// TIA Portal V16 export
// export: Created 2024-12-03T15:41:45.7340631Z, ExportSetting WithReadOnly, DisplayName Totally Integrated Automation Portal, DisplayVersion V16 Update 6, DisplayName TIA Portal Version Control Interface, DisplayVersion V16 Update 2, DisplayName TIA Portal Openness, DisplayVersion V16 Update 6, DisplayName TIA Portal Teamcenter Gateway, DisplayVersion V16, DisplayName SINAMICS Startdrive Advanced, DisplayVersion V16 Update 5, DisplayName SINAMICS Startdrive G130, G150, S120, S150, SINAMICS MV, S210, DisplayVersion V16 Update 5, DisplayName SINAMICS Startdrive G110M, G120, G120C, G120D, G120P, G115D, DisplayVersion V16 Update 5, DisplayName STEP 7 Professional, DisplayVersion V16 Update 6, DisplayName STEP 7 Safety, DisplayVersion V16, DisplayName WinCC Advanced / Unified PC, DisplayVersion V16 Update 6
TYPE "Nord_Drive_UDT"
// stored: CreationDate 2023-04-19T11:30:38.0051651Z, InterfaceModifiedDate 2023-04-19T12:03:36.1263348Z, IsConsistent true, LibraryConformanceStatus The object is library-conformant., ModifiedDate 2023-04-19T12:03:36.1263348Z
   STRUCT
      Cmd : Struct   // MotorCommands
         Reset : Bool;
         OnAuto : Bool;
         OnManual : Bool;
         DirectionAuto : Bool;
         DirectionManual : Bool;
         SpeedAuto : Real;
         SpeedManual : Real;
         Interlock : Bool;
      END_STRUCT;
      Alarms : Struct
         NotOnTImedOut : "HmiAlarm";   // Motor not on in time
         NotOffTimedOut : "HmiAlarm";   // Motor not off in time
         ErrorFromDrive : "HmiAlarm";   // Error from drive
         CannotStartError : "HmiAlarm";   // Cannot start error
         EmergencyStopActive : "HmiAlarm";   // Emergency stop is active
         Disconnected : "HmiAlarm";   // The device is not connected
         WarningFromDrive { S7_SetPoint := 'True'} : "HmiAlarm";   // Warning from drive
         AlarmStatus : Word;   // lsb 0 not on | lsb 1 not off | lsb 2 error from drive | lsb 3 cannot start | 4 emergency stop active | 5 disconnected
      END_STRUCT;
      Status : Struct
         CmdRunManualActive : Bool;
         Interlocked : Bool;
         ManualModeActive : Bool;
         ManualCommandsDisabled : Bool;
         Running : Bool;
         ActualSpeed : Real;
         ActualDirection : Bool;   // 0 right | 1 left
         ReadyToStart : Bool;
         ReadyForOperaiton : Bool;
         PowerOn : Bool;
         Status : Word;   // lsb 0 interlocked | lsb 1 running | lbs2 manual mode active | lsb3 warning active on drive | lsb4 readyTostart | lsb5 ready for operation | lsb6 powered
      END_STRUCT;
      Settings : Struct
         DefaultDirection : Bool;
         InverseDirectionLabel : Bool;
         AllowManualDirection : Bool;
         MaxSpeedManual : Real;
         MinSpeedManual : Real;
      END_STRUCT;
      Zone : Int;
      Commonstatus : Int;
      GroupNumber : Int;
      info : "MotorInfo";
   END_STRUCT;
END_TYPE
